// TwinCAT 3 PLC project PLC_Ladder_Hardware_Integration
// ProgramVersion: 3.1.4024.0
// CompilerDefines: VISU_USEWSTRING
// libraries:
//   Tc2_Math, * (Beckhoff Automation GmbH)
//   Tc2_MC2, * (Beckhoff Automation GmbH)
//   Tc2_NC, * (Beckhoff Automation GmbH)
//   Tc2_Standard, * (Beckhoff Automation GmbH)
//   Tc2_System, * (Beckhoff Automation GmbH)
//   Tc2_Utilities, * (Beckhoff Automation GmbH)
//   Tc3_Module, * (Beckhoff Automation GmbH)
// project tree:
//   / GlobalTextList.TcGTLO (not stored), PlcTask.TcTTO, Visualization Manager.TcVMO (not stored), VISU_TASK.TcTTO
//   GVLs/ GVL.TcGVL, GVLLD.TcGVL
//   POUs/ MAIN.TcPOU, ladder_logic_diagram.TcPOU, Meters_Travelled.TcPOU (not stored), SYSTEM.TcPOU, Safety_Zones.TcDUT (not stored), TP_and_TON_For_timeout.TcPOU
//   VISUs/ Charge_Velocity_Distance.TcVIS (not stored), Header.TcVIS (not stored), ImagePool.TcIPO (not stored), log_file.TcVIS (not stored), MainScreen.TcVIS (not stored), Nav.TcVIS (not stored), Nav_1.TcVIS (not stored), Safty_Zones_and_Modes.TcVIS (not stored)
// real-time tasks:
//   TASK PlcTask: cycle T#10ms, priority 20, ADS port 350
//   TASK VISU_TASK: cycle T#200000us, priority 30, ADS port 351
// motion (NC):
//   TASK NC-Task 1 SAF: cycle T#2ms, priority 4, ADS port 501
//   TASK NC-Task 1 SVB: cycle T#10ms, priority 8, ADS port 511
//   AXIS Axis 1 (id 1)
//     Dynamic: Acceleration=2181.51, Deceleration=2181.51, Jerk=6544.55
//     Velo: RefSearch=14.5434333333333, RefSync=14.5434333333333, SlowManual=72.7171666666667, FastManual=436.303, Fast=1454.34333333333, Maximum=1454.34
//     TargetPosControl: Range=20
//     OtherSettings: AllowMotionCmdToSlave=true
//     encoder EncType=19
//       EncPara: ScaleFactorNumerator=15.7, ScaleFactorDenominator=1048576, MaxCount=#xffffffff
//     drive DrvType=16
//       DrvPara: MaxCount=#xffffffff
//         Analog: VeloReferenz=1599.77766666667, VeloScale=32, TorqueSetpointScale=10, ScaleFactorActTorque=0.1
//         TimeComp: TaskDelayCycles=1
//     controller CtrType=1
//       CtrPara: PriorControlFactor=1
//         PosDiffControl: Range=40000
//         Observer: BandWidth=20
//   AXIS Axis 2 (id 2)
//     Dynamic: Acceleration=2181.515, Deceleration=2181.515, Jerk=6544.545
//     Velo: RefSearch=14.5434333333333, RefSync=14.5434333333333, SlowManual=72.7171666666667, FastManual=436.303, Fast=1454.34333333333, Maximum=1454.34333333333
//     TargetPosControl: Range=20
//     OtherSettings: AllowMotionCmdToSlave=true
//     encoder EncType=19
//       EncPara: ScaleFactorNumerator=15.7, ScaleFactorDenominator=1048576, MaxCount=#xffffffff
//     drive DrvType=16
//       DrvPara: MaxCount=#xffffffff
//         Analog: VeloReferenz=1599.77766666667, VeloScale=32, TorqueSetpointScale=10, ScaleFactorActTorque=0.1
//         TimeComp: TaskDelayCycles=1
//     controller CtrType=1
//       CtrPara: PriorControlFactor=1
//         PosDiffControl: Range=40000
//         Observer: BandWidth=20
//   AXIS Axis 3 (id 3)
//     Dynamic: Acceleration=8031.31, Deceleration=8031.31, Jerk=24093.9
//     Velo: RefSearch=53.5420666666667, RefSync=53.5420666666667, SlowManual=267.710333333333, FastManual=1606.262, Fast=5354.20666666667, Maximum=5354.21
//     OtherSettings: AllowMotionCmdToSlave=true
//     encoder EncType=19
//       EncPara: ScaleFactorNumerator=57.8, ScaleFactorDenominator=1048576, MaxCount=#xffffffff
//     drive DrvType=16
//       DrvPara: MaxCount=#xffffffff
//         Analog: VeloReferenz=5889.62733333333, VeloScale=32, TorqueSetpointScale=10, ScaleFactorActTorque=0.1
//         TimeComp: TaskDelayCycles=1
//     controller CtrType=1
//       CtrPara: PriorControlFactor=1
//         PosDiffControl: Range=4000
//         Observer: BandWidth=20
// variable links:
//   PLC_Ladder_Hardware_Integration/PLC_Ladder_Hardware_Integration Instance <-> NC-Task 1 SAF/Axes/Axis 1
//     PlcTask Inputs/MAIN.AxisB.NcToPlc <-> Outputs/ToPlc
//     PlcTask Outputs/MAIN.AxisB.PlcToNc <-> Inputs/FromPlc
//   PLC_Ladder_Hardware_Integration/PLC_Ladder_Hardware_Integration Instance <-> NC-Task 1 SAF/Axes/Axis 2
//     PlcTask Inputs/MAIN.AxisA.NcToPlc <-> Outputs/ToPlc
//     PlcTask Outputs/MAIN.AxisA.PlcToNc <-> Inputs/FromPlc

CONFIGURATION PLC_Ladder_Hardware_Integration
    RESOURCE PLC ON TwinCAT3
        TASK PlcTask(INTERVAL := T#10ms, PRIORITY := 20);
        TASK VISU_TASK(INTERVAL := T#200000us, PRIORITY := 30);
        PROGRAM MAIN WITH PlcTask : MAIN;
        PROGRAM VisuElems_Visu_Prg WITH VISU_TASK : VisuElems.Visu_Prg;
    END_RESOURCE
END_CONFIGURATION

// ---- GVLs/GVL.TcGVL
{attribute 'qualified_only'}
VAR_GLOBAL
	
	GetLocalSystemTime : FB_LocalSystemTime;
	SystemDateTime : STRING;
	SystemDate : STRING;
	SystemTime : STRING;
	SystemSeconds : STRING;
END_VAR

// ---- GVLs/GVLLD.TcGVL
{attribute 'qualified_only'}
VAR_GLOBAL
	
//Input Variables 
ONOFF_Buton               AT %I* : BOOL;
Manual_Stop_Buton         AT %I* : BOOL;
Manual_Mode_Buton         AT %I* : BOOL;
Autonomous_Mode_Buton     AT %I* : BOOL;
Lock_Mode_Buton           AT %I* : BOOL;
Clear_Reset_Buton         AT %I* : BOOL;
Resume_Buton              AT %I* : BOOL;
view_safety               AT %I* : BOOL;


//Output Variables 
Brake                     AT %Q* : BOOL;  
Kontak                    AT %Q* : BOOL;
Front_White_Zone          AT %Q* : BOOL;
Front_Red_Zone            AT %Q* : BOOL;
Front_Purple_Zone         AT %Q* : BOOL;
Front_Grey_Pink_Zone      AT %Q* : BOOL;
Robot_Clear_Lidar         AT %Q* : BOOL;
Robot_Manual_Mode         AT %Q* : BOOL;
Robot_Autonomous_Mode     AT %Q* : BOOL;
Robot_Lock_Mode           AT %Q* : BOOL;
Robot_Mode_Run            AT %Q* : BOOL;
lift_up_Q                 AT %Q* : BOOL;
lift_down_Q            	  AT %Q* : BOOL;
zone_1                    AT %Q* : BOOL;
zone_2                    AT %Q* : BOOL;
zone_3                    AT %Q* : BOOL;
zone_4                    AT %Q* : BOOL;
zone_5                    AT %Q* : BOOL;
zone_6                    AT %Q* : BOOL;
auto_charge_signal        AT %Q* : BOOL;

//Memery Variables 

System_Trig               AT %M* : BOOL;
System_Set                AT %M* : BOOL;
Memory_Set		          AT %M* : BOOL;
White                     AT %M* : BOOL;
Red                       AT %M* : BOOL;
Purple                    AT %M* : BOOL;
Grey_Pink                 AT %M* : BOOL;
Lock_Mode_Reset           AT %M* : BOOL;
lift_up           		  AT %M* : BOOL;
lift_down				  AT %M* : BOOL;
lift_stop				  AT %M* : BOOL;
elavator_up				  AT %M* : BOOL;
elavator_down			  AT %M* : BOOL;
auto_charge_on            AT %M* : BOOL;
auto_charge_off           AT %M* : BOOL;
view_safety_state         AT %M* : BOOL;

first_read		          AT %M* : BOOL;
second_read               AT %M* : BOOL;








	real_trigger: BOOL;
END_VAR

// ---- POUs/MAIN.TcPOU
PROGRAM MAIN
VAR
	Lidar_zones:  Safety_Zones; 
	encoderPosition AT  %I* : UDINT;
	actualAxisPosition AT  %I* : LREAL;
	actualAxisPositionA AT  %I* : LREAL;
	Left_Encoder : LREAL;
	Right_Encoder : LREAL;
	setPositionA AT  %I* : LREAL ;
	setPositionB AT  %I* : LREAL ;
	AxisB : AXIS_REF; //left Motor
	AxisA : AXIS_REF; //Right Motor
	AxisC : AXIS_REF; //Roller Axis
	timer : TON;
	// Motor 1
	McPower : MC_Power;
	McReset : MC_Reset;
	McJogging : MC_Jog;
	McVelocity : MC_MoveVelocity;
	McStop :  MC_Stop;
	McHalt : MC_Halt;
	McSetPositionA: MC_SetPosition;
	McSetPosition: MC_SetPosition;
	McPosition : MC_ReadActualPosition;
	McPositionA : MC_ReadActualPosition;
	McRelativeVelocity : MC_MoveRelative;
	

	// Motor 2
	McPowerA : MC_Power;
	McResetA : MC_Reset;
	McJoggingA : MC_Jog;
	McVelocityA : MC_MoveVelocity;
	McStopA :  MC_Stop;
	McHaltA : MC_Halt;
	
	CppVelocityValue : DINT;
	CppVelocityCmd : DINT;
	RightVelocityValue : REAL;
	LeftVelocityValue : REAL;
	RightVelocityCmd : REAL;
	LeftVelocityCmd : REAL;
	RollerVelocityValue : REAL;
	RollerVelocityCmd : REAL;
	RightVelocity_meters : REAL;
	LeftVelocity_meters : REAL;
	acc : REAL:=0;
	dcc : REAL:=0;
	jk	: REAL:=0;
	myvelocity : DINT;
	cppvar AT %I* : BOOL;
	pypositive AT %I* : BOOL;
	pynegative AT %I* : BOOL;
	pyturnright AT %I* : BOOL;
	pyturnleft AT %I* : BOOL;
	state : DINT;
	stop AT %I* : BOOL;
	fright AT %I* : BOOL;
	bright AT %I* : BOOL;
	fleft AT %I* : BOOL;
	bleft AT %I* : BOOL;
	roller_forward     AT %I* : BOOL;
	roller_backwrad    AT %I* : BOOL;
	ChargeSignal       AT %Q* : BOOL;
	Lift_UP            AT %Q* : BOOL:= FALSE;
	Lift_DOWN          AT %Q* : BOOL;
	Lift_UP_Signal	   AT %M* : BOOL;
	Lift_DOWN_Signal   AT %M* : BOOL;
	Lift_Stop          AT %M* : BOOL;
	FrontLidarWarning  AT %I* : BOOL;
	BackLidarWarning   AT %I* : BOOL;

	stopvalue : BOOL;
	Acceleration: LREAL;
	Options: INT;
	nVAR: REAL;
	
	time_first_read : INT;
	time_second_read : INT;
	//Lidar Zones
	zon_1_set          AT %M* : BOOL; 
	zon_2_set          AT %M* : BOOL; 
	zon_3_set          AT %M* : BOOL; 
	zon_4_set          AT %M* : BOOL; 
	zon_5_set          AT %M* : BOOL; 
	zon_6_set          AT %M* : BOOL;    
	
	
	
END_VAR

SYSTEM();
Meters_Travelled();
Ladder_Logic_Diagram();
encoderPosition;
TP_and_TON_For_timeout();

IF GVLLD.first_read THEN	
time_first_read := STRING_TO_INT (GVL.SystemSeconds);
END_IF
IF GVLLD.second_read THEN	
time_second_read := STRING_TO_INT (GVL.SystemSeconds);
END_IF

// Axis B Left Motor
AxisB.ReadStatus();
McPower(Axis:=AxisB,Enable := TRUE,Enable_Positive := TRUE, Enable_Negative := TRUE);
McSetPosition(Axis:= AxisB,Execute:= TRUE, Position := setPositionA);
McPosition(Axis := AxisB,Enable := TRUE );
actualAxisPosition := McPosition.Position;
Left_Encoder := actualAxisPosition ;

// Axis A Right Motor
AxisA.ReadStatus();
McPowerA(Axis:=AxisA,Enable := TRUE,Enable_Positive := TRUE, Enable_Negative := TRUE);
McSetPositionA(Axis:= AxisA,Execute:= TRUE, Position := setPositionB);
McPositionA(Axis := AxisA,Enable := TRUE );
actualAxisPositionA := McPositionA.Position;
Right_Encoder := actualAxisPositionA ;


CppVelocityCmd := CppVelocityValue;
RightVelocity_meters := RightVelocityCmd /1000 ;
LeftVelocity_meters := LeftVelocityCmd / 1000 ;
IF NOT GVLLD.view_safety THEN
	RightVelocityCmd := 0;
	LeftVelocityCmd := 0;
	RollerVelocityCmd := 0;
	ELSE IF NOT FrontLidarWarning OR NOT BackLidarWarning THEN
		RightVelocityCmd := RightVelocityValue * 0.9;
		LeftVelocityCmd := LeftVelocityValue * 0.9;
	ELSE IF FrontLidarWarning OR BackLidarWarning THEN
		RightVelocityCmd := RightVelocityValue;
		LeftVelocityCmd := LeftVelocityValue;
		RollerVelocityCmd := RollerVelocityValue;
		END_IF
	END_IF
END_IF

stopvalue := stop;



CASE state OF 
	0: 	
		state := 10;
	10: 
	
		McReset(Axis := AxisB,Execute := TRUE);
		McResetA(Axis := AxisA,Execute := TRUE);
		IF McReset.Done AND McResetA.Done  THEN
			state := 20;
		ELSIF NOT McReset.Done OR NOT McResetA.Done THEN 
			McReset(Axis := AxisB,Execute := FALSE);
			McResetA(Axis := AxisA,Execute := FALSE);
			McReset(Axis := AxisB,Execute := TRUE);
			McResetA(Axis := AxisA,Execute := TRUE);
			state := 20;
		END_IF
		
	20: 
	
		McPowerA(Axis:=AxisA,Enable := TRUE,Enable_Positive := TRUE, Enable_Negative := TRUE);
		McPower(Axis:=AxisB,Enable := TRUE,Enable_Positive := TRUE, Enable_Negative := TRUE);
		IF McPower.Status AND McPowerA.Status THEN
			McReset(Axis := AxisB,Execute := TRUE);
			McResetA(Axis := AxisA,Execute := TRUE);
			IF McReset.Done AND McResetA.Done  THEN
				state :=50;
			ELSIF NOT McReset.Done OR NOT McResetA.Done THEN 
				McReset(Axis := AxisB,Execute := FALSE);
				McResetA(Axis := AxisA,Execute := FALSE);
				McReset(Axis := AxisB,Execute := TRUE);
				McResetA(Axis := AxisA,Execute := TRUE);
				state :=50;
			END_IF
		END_IF
		
	
	//CPP Function Block
//	40: 
		
//		McVelocityA (Axis:= AxisA,
//					Execute := cppvar,
//					Velocity := CppVelocityCmd,
//						Acceleration := acc,
//						Deceleration := dcc,
//						Jerk := jk,
//					Direction := MC_Direction.MC_Positive_Direction ) ;
//		McVelocity (Axis:= AxisB,
//					Execute := cppvar,
//					Velocity := CppVelocityCmd,
//						Acceleration := acc,
//						Deceleration := dcc,
//						Jerk := jk,
//					Direction := MC_Direction.MC_Positive_Direction ) ;
//		McVelocityA (Axis:= AxisA,
//					Execute := cppvar,
//					Velocity := CppVelocityCmd,
//						Acceleration := acc,
//						Deceleration := dcc,
//						Jerk := jk,
//					Direction := MC_Direction.MC_Negative_Direction ) ;
//		McVelocity (Axis:= AxisB,
//					Execute := cppvar,
//					Velocity := CppVelocityCmd,
//						Acceleration := acc,
//						Deceleration := dcc,
//						Jerk := jk,
//					Direction := MC_Direction.MC_Negative_Direction ) ;
//		IF stopvalue THEN
//			McVelocity(Axis := AxisB, Execute := FALSE); 
//			McVelocityA(Axis := AxisA, Execute := FALSE); 
//			state := 900;
//		END_IF
//		IF fright OR fleft OR bright OR bleft THEN 
//			McVelocity(Axis := AxisB, Execute := FALSE);
//			McVelocityA(Axis := AxisA, Execute := FALSE);
//			state := 50;
//		END_IF
		
		
	//Python Function Block
	50: 
		// POSİTİVE
		IF AxisA.Status.Error OR AxisB.Status.Error THEN 
			McReset(Axis := AxisB,Execute := FALSE);
			McResetA(Axis := AxisA,Execute := FALSE);
			McReset(Axis := AxisB,Execute := TRUE);
			McResetA(Axis := AxisA,Execute := TRUE);
//			state :=0;
		END_IF
		IF stopvalue THEN
			
			McVelocity(Axis := AxisB, Execute := FALSE); 
			McVelocityA(Axis := AxisA, Execute := FALSE);
			state := 900;
		END_IF
		IF GVLLD.auto_charge_signal THEN   
   			McVelocity(Axis := AxisB, Execute := FALSE);    
			McVelocityA(Axis := AxisA, Execute := FALSE);
  			state := 400;  
		END_IF
		
		McVelocityA (Axis:= AxisA,
						Execute := fright,
						Velocity := RightVelocityCmd,
						Acceleration := acc,
						Deceleration := dcc,
						Jerk := jk,
						Direction := MC_Direction.MC_Positive_Direction ) ;
		McVelocityA (Axis:= AxisA,
						Execute := bright,
						Velocity := RightVelocityCmd,
						Acceleration := acc,
						Deceleration := dcc,
						Jerk := jk,
						Direction := MC_Direction.MC_Negative_Direction ) ;
		McVelocity (Axis:= AxisB,
						Execute := fleft,
						Velocity := LeftVelocityCmd,
						Acceleration := acc,
						Deceleration := dcc,
						Jerk := jk,
						Direction := MC_Direction.MC_Positive_Direction ) ;
		McVelocity (Axis:= AxisB,
						Execute := bleft,
						Velocity := LeftVelocityCmd,
						Acceleration := acc,
						Deceleration := dcc,
						Jerk := jk,
						Direction := MC_Direction.MC_Negative_Direction ) ;
// Roller Velocity Blocks
//Forward
//		MC_MoveContinuousRelative(Axis:=AxisC,
//								Execute:= roller_forward,
//								Distance:= 5000,
//								Velocity:= 1000,
//								EndVelocity:= 0,
//								Acceleration:= acc,
//								Deceleration:= dcc,
//								Jerk:= jk);
////Backward 
//		MC_MoveContinuousRelative(Axis:=AxisC,
//								Execute:= roller_backwrad,
//								Distance:= 5000,
//								Velocity:= RollerVelocityValue,
//								EndVelocity:= 0,
//								Acceleration:= acc,
//								Deceleration:= dcc,
//								Jerk:= jk);
		IF cppvar THEN 
			McVelocity(Axis := AxisB, Execute := FALSE);
			McVelocityA(Axis := AxisA, Execute := FALSE);
			state := 40;
		END_IF
	400:  
		IF AxisA.Status.Error OR AxisB.Status.Error THEN 
		   	McReset(Axis := AxisB,Execute := FALSE);   
			McResetA(Axis := AxisA,Execute := FALSE);
		   	McReset(Axis := AxisB,Execute := TRUE);   
			McResetA(Axis := AxisA,Execute := TRUE);
  		END_IF
    	McStop(Axis := AxisB, Execute := TRUE);
  		McStopA(Axis := AxisA, Execute := TRUE);  
  		IF NOT GVLLD.auto_charge_signal THEN   
			McStop(Axis := AxisB, Execute := FALSE); 
			McVelocity(Axis := AxisB, Execute := FALSE);    
			McStopA(Axis := AxisA, Execute := FALSE); 
			McVelocityA(Axis := AxisA, Execute := FALSE);    
			state := 50;
  		END_IF
	900:
		IF AxisA.Status.Error OR AxisB.Status.Error THEN 
			McReset(Axis := AxisB,Execute := FALSE);
			McResetA(Axis := AxisA,Execute := FALSE);
			McReset(Axis := AxisB,Execute := TRUE);
			McResetA(Axis := AxisA,Execute := TRUE);
		END_IF
		McStop(Axis := AxisB, Execute := TRUE);
		McStopA(Axis := AxisA, Execute := TRUE);
		IF fright OR fleft OR bright OR bleft OR pyturnleft OR cppvar THEN
			McStop(Axis := AxisB, Execute := FALSE); 
			McVelocity(Axis := AxisB, Execute := FALSE); 
			McStopA(Axis := AxisA, Execute := FALSE); 
			McVelocityA(Axis := AxisA, Execute := FALSE); 
			state := 50;
		END_IF
		
		
		
END_CASE

END_PROGRAM

// ---- POUs/SYSTEM.TcPOU
PROGRAM SYSTEM
VAR
END_VAR

GVL.GetLocalSystemTime(
	sNetID := ,
	bEnable := TRUE,
	dwCycle := 1,
	dwOpt:= ,
	tTimeout:= ,
	bValid =>,
	systemTime=>,
	tzID=>);
	
GVL.SystemDateTime := SYSTEMTIME_TO_STRING(GVL.GetLocalSystemTime.systemTime);
GVL.SystemDate := MID(STR:= GVL.SystemDateTime,LEN:=10,POS:=1);
GVL.SystemTime := MID(STR:= GVL.SystemDateTime,LEN:=8,POS:=12);
GVL.SystemSeconds := MID(STR:= GVL.SystemDateTime,LEN:=2,POS:=18);

END_PROGRAM

// ---- POUs/ladder_logic_diagram.TcPOU
PROGRAM ladder_logic_diagram 
VAR
	t2s: TIME := TIME#3S;
	t0s: TIME := TIME#0S;
	Timer: TON;
	input : BOOL;
	output : BOOL; 
	TON_Reset: TON;
	TON_set: TON;
	TON_0: TON;
	TON_Trig: TON;
	TON_Autonomous: TON;
	TON_Manual: TON;
	TON_Lock: TON;
	Robot_Mode_Timer: TON;
	liftUP: TON;
	liftDOWN: TON;

	T: TIME;
	Activate_time_read: BOOL;
	TON_1: TON;
	first_read_triggerd: BOOL;
	TON_2: TON;
	second_read_triggerd: BOOL;
	TON_3: TON;
	TON_4: TON;
	TON_5: TON;
	trig_1: BOOL;
	TP_0: TP;
	TP_1: TP;
	trig_2: BOOL;
	load_button: BOOL;
	TON_6: TON;
	load_active: BOOL;
	TON_7: TON;
END_VAR
VAR // added by the converter: edge detectors and wires of the graphical bodies
    _rt1 : R_TRIG;
    _w1 : BOOL;
END_VAR

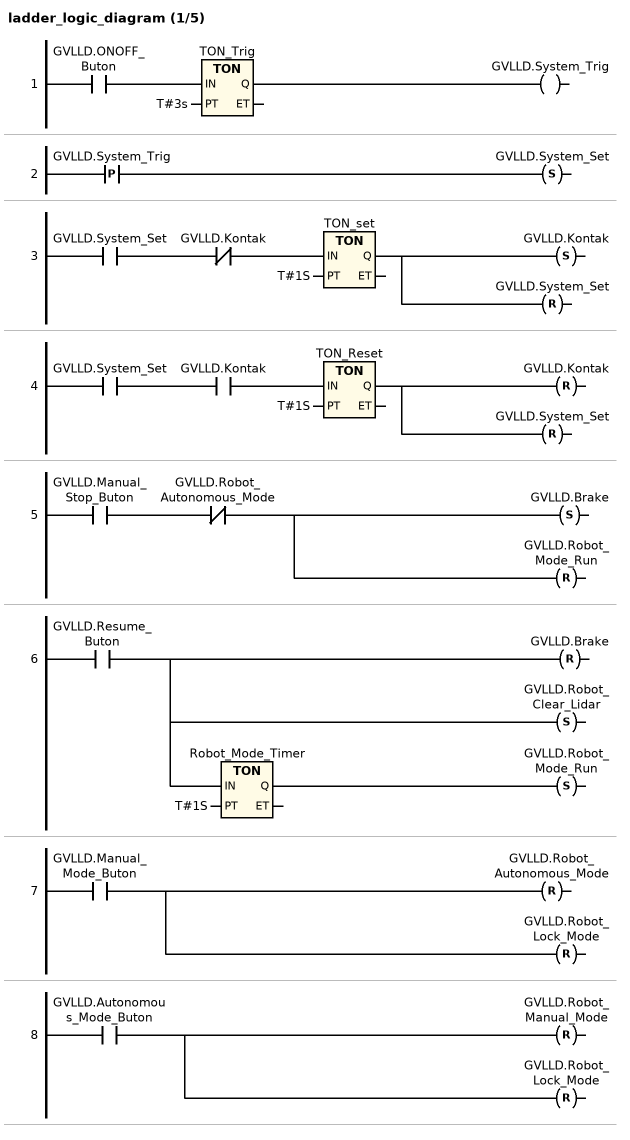
// NETWORK 1
TON_Trig(IN := GVLLD.ONOFF_Buton, PT := T#3s); // TON
GVLLD.System_Trig := TON_Trig.Q;

// NETWORK 2
_rt1(CLK := GVLLD.System_Trig);
GVLLD.System_Set S= _rt1.Q;

// NETWORK 3
TON_set(IN := GVLLD.System_Set AND NOT GVLLD.Kontak, PT := T#1S); // TON
GVLLD.Kontak S= TON_set.Q;
GVLLD.System_Set R= TON_set.Q;

// NETWORK 4
TON_Reset(IN := GVLLD.System_Set AND GVLLD.Kontak, PT := T#1S); // TON
GVLLD.Kontak R= TON_Reset.Q;
GVLLD.System_Set R= TON_Reset.Q;

// NETWORK 5
_w1 := GVLLD.Manual_Stop_Buton AND NOT GVLLD.Robot_Autonomous_Mode;
GVLLD.Brake S= _w1;
GVLLD.Robot_Mode_Run R= _w1;

// NETWORK 6
GVLLD.Brake R= GVLLD.Resume_Buton;
GVLLD.Robot_Clear_Lidar S= GVLLD.Resume_Buton;
Robot_Mode_Timer(IN := GVLLD.Resume_Buton, PT := T#1S); // TON
GVLLD.Robot_Mode_Run S= Robot_Mode_Timer.Q;

// NETWORK 7
GVLLD.Robot_Autonomous_Mode R= GVLLD.Manual_Mode_Buton;
GVLLD.Robot_Lock_Mode R= GVLLD.Manual_Mode_Buton;

// NETWORK 8
GVLLD.Robot_Manual_Mode R= GVLLD.Autonomous_Mode_Buton;
GVLLD.Robot_Lock_Mode R= GVLLD.Autonomous_Mode_Buton;

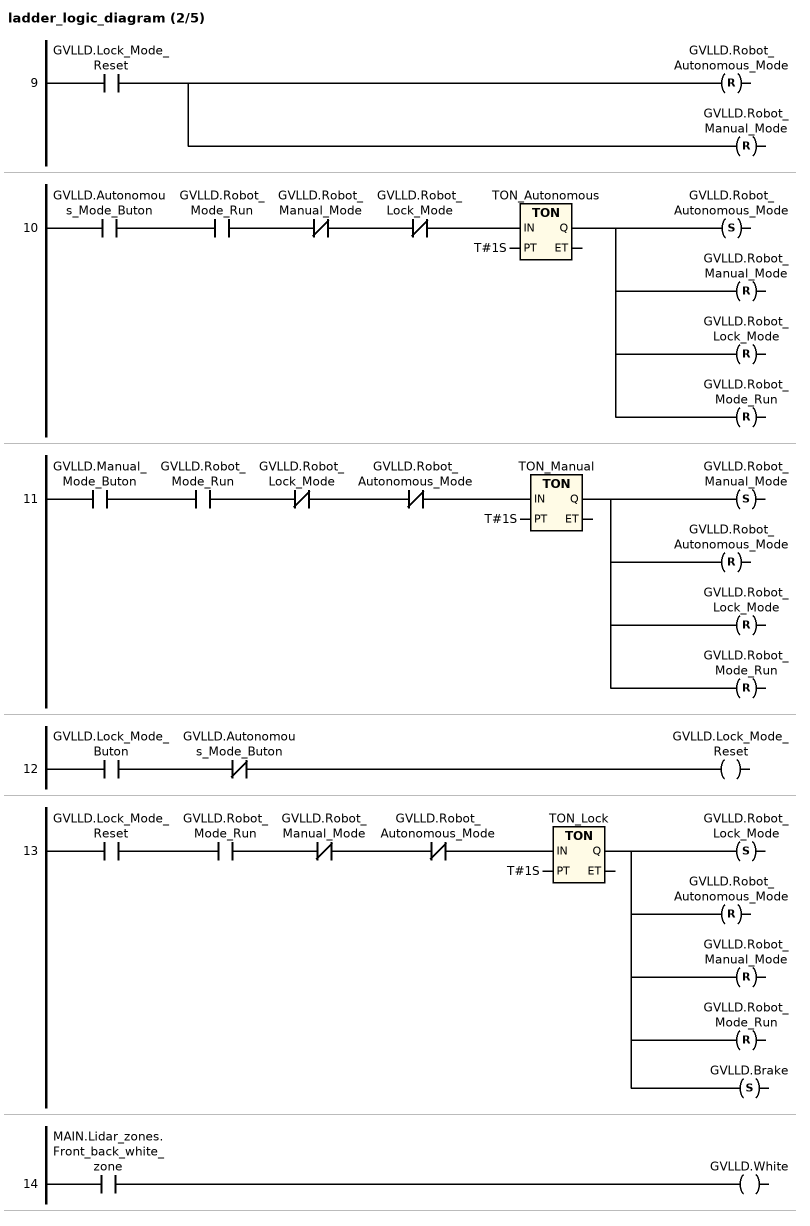
// NETWORK 9
GVLLD.Robot_Autonomous_Mode R= GVLLD.Lock_Mode_Reset;
GVLLD.Robot_Manual_Mode R= GVLLD.Lock_Mode_Reset;

// NETWORK 10
TON_Autonomous(IN := GVLLD.Autonomous_Mode_Buton AND GVLLD.Robot_Mode_Run AND NOT GVLLD.Robot_Manual_Mode AND NOT GVLLD.Robot_Lock_Mode, PT := T#1S); // TON
GVLLD.Robot_Autonomous_Mode S= TON_Autonomous.Q;
GVLLD.Robot_Manual_Mode R= TON_Autonomous.Q;
GVLLD.Robot_Lock_Mode R= TON_Autonomous.Q;
GVLLD.Robot_Mode_Run R= TON_Autonomous.Q;

// NETWORK 11
TON_Manual(IN := GVLLD.Manual_Mode_Buton AND GVLLD.Robot_Mode_Run AND NOT GVLLD.Robot_Lock_Mode AND NOT GVLLD.Robot_Autonomous_Mode, PT := T#1S); // TON
GVLLD.Robot_Manual_Mode S= TON_Manual.Q;
GVLLD.Robot_Autonomous_Mode R= TON_Manual.Q;
GVLLD.Robot_Lock_Mode R= TON_Manual.Q;
GVLLD.Robot_Mode_Run R= TON_Manual.Q;

// NETWORK 12
GVLLD.Lock_Mode_Reset := GVLLD.Lock_Mode_Buton AND NOT GVLLD.Autonomous_Mode_Buton;

// NETWORK 13
TON_Lock(IN := GVLLD.Lock_Mode_Reset AND GVLLD.Robot_Mode_Run AND NOT GVLLD.Robot_Manual_Mode AND NOT GVLLD.Robot_Autonomous_Mode, PT := T#1S); // TON
GVLLD.Robot_Lock_Mode S= TON_Lock.Q;
GVLLD.Robot_Autonomous_Mode R= TON_Lock.Q;
GVLLD.Robot_Manual_Mode R= TON_Lock.Q;
GVLLD.Robot_Mode_Run R= TON_Lock.Q;
GVLLD.Brake S= TON_Lock.Q;

// NETWORK 14
GVLLD.White := MAIN.Lidar_zones.Front_back_white_zone;

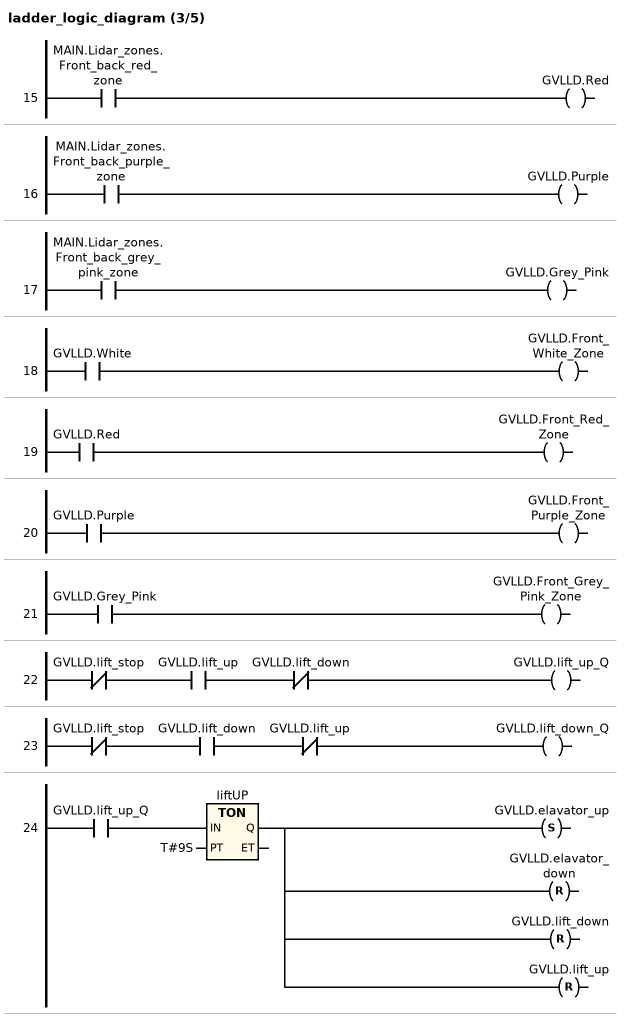
// NETWORK 15
GVLLD.Red := MAIN.Lidar_zones.Front_back_red_zone;

// NETWORK 16
GVLLD.Purple := MAIN.Lidar_zones.Front_back_purple_zone;

// NETWORK 17
GVLLD.Grey_Pink := MAIN.Lidar_zones.Front_back_grey_pink_zone;

// NETWORK 18
GVLLD.Front_White_Zone := GVLLD.White;

// NETWORK 19
GVLLD.Front_Red_Zone := GVLLD.Red;

// NETWORK 20
GVLLD.Front_Purple_Zone := GVLLD.Purple;

// NETWORK 21
GVLLD.Front_Grey_Pink_Zone := GVLLD.Grey_Pink;

// NETWORK 22
GVLLD.lift_up_Q := NOT GVLLD.lift_stop AND GVLLD.lift_up AND NOT GVLLD.lift_down;

// NETWORK 23
GVLLD.lift_down_Q := NOT GVLLD.lift_stop AND GVLLD.lift_down AND NOT GVLLD.lift_up;

// NETWORK 24
liftUP(IN := GVLLD.lift_up_Q, PT := T#9S); // TON
GVLLD.elavator_up S= liftUP.Q;
GVLLD.elavator_down R= liftUP.Q;
GVLLD.lift_down R= liftUP.Q;
GVLLD.lift_up R= liftUP.Q;

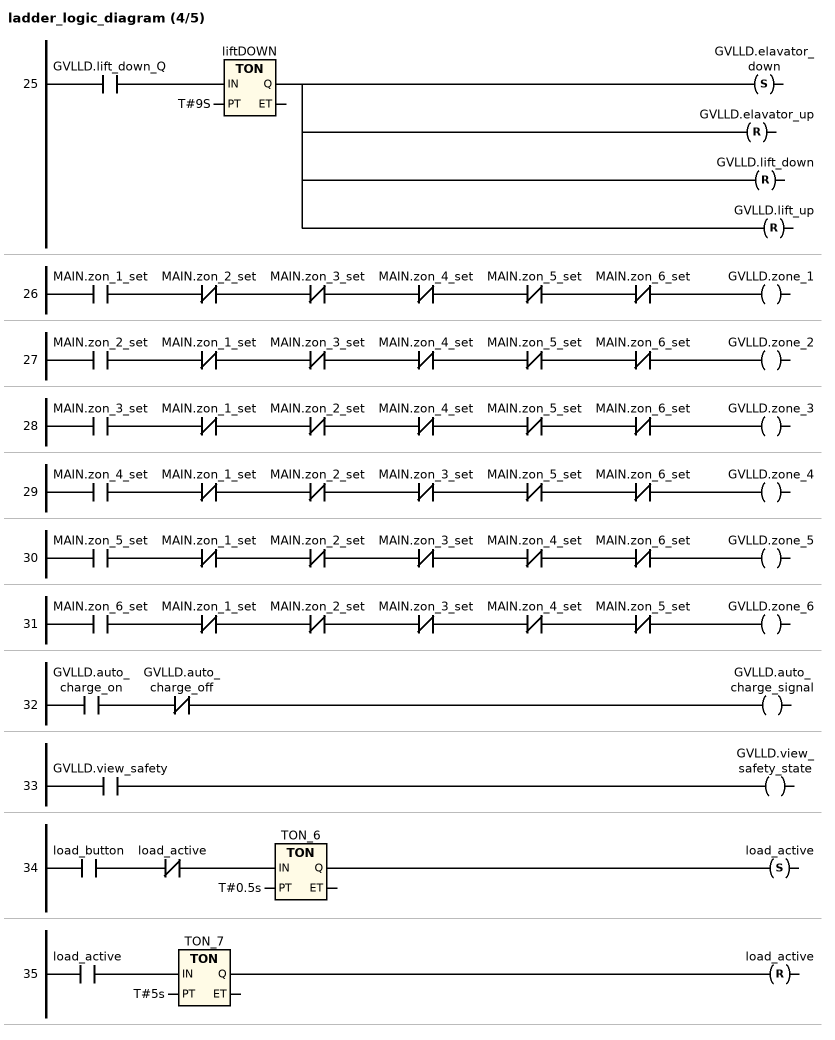
// NETWORK 25
liftDOWN(IN := GVLLD.lift_down_Q, PT := T#9S); // TON
GVLLD.elavator_down S= liftDOWN.Q;
GVLLD.elavator_up R= liftDOWN.Q;
GVLLD.lift_down R= liftDOWN.Q;
GVLLD.lift_up R= liftDOWN.Q;

// NETWORK 26
GVLLD.zone_1 := MAIN.zon_1_set AND NOT MAIN.zon_2_set AND NOT MAIN.zon_3_set AND NOT MAIN.zon_4_set AND NOT MAIN.zon_5_set AND NOT MAIN.zon_6_set;

// NETWORK 27
GVLLD.zone_2 := MAIN.zon_2_set AND NOT MAIN.zon_1_set AND NOT MAIN.zon_3_set AND NOT MAIN.zon_4_set AND NOT MAIN.zon_5_set AND NOT MAIN.zon_6_set;

// NETWORK 28
GVLLD.zone_3 := MAIN.zon_3_set AND NOT MAIN.zon_1_set AND NOT MAIN.zon_2_set AND NOT MAIN.zon_4_set AND NOT MAIN.zon_5_set AND NOT MAIN.zon_6_set;

// NETWORK 29
GVLLD.zone_4 := MAIN.zon_4_set AND NOT MAIN.zon_1_set AND NOT MAIN.zon_2_set AND NOT MAIN.zon_3_set AND NOT MAIN.zon_5_set AND NOT MAIN.zon_6_set;

// NETWORK 30
GVLLD.zone_5 := MAIN.zon_5_set AND NOT MAIN.zon_1_set AND NOT MAIN.zon_2_set AND NOT MAIN.zon_3_set AND NOT MAIN.zon_4_set AND NOT MAIN.zon_6_set;

// NETWORK 31
GVLLD.zone_6 := MAIN.zon_6_set AND NOT MAIN.zon_1_set AND NOT MAIN.zon_2_set AND NOT MAIN.zon_3_set AND NOT MAIN.zon_4_set AND NOT MAIN.zon_5_set;

// NETWORK 32
GVLLD.auto_charge_signal := GVLLD.auto_charge_on AND NOT GVLLD.auto_charge_off;

// NETWORK 33
GVLLD.view_safety_state := GVLLD.view_safety;

// NETWORK 34
TON_6(IN := load_button AND NOT load_active, PT := T#0.5s); // TON
load_active S= TON_6.Q;

// NETWORK 35
TON_7(IN := load_active, PT := T#5s); // TON
load_active R= TON_7.Q;

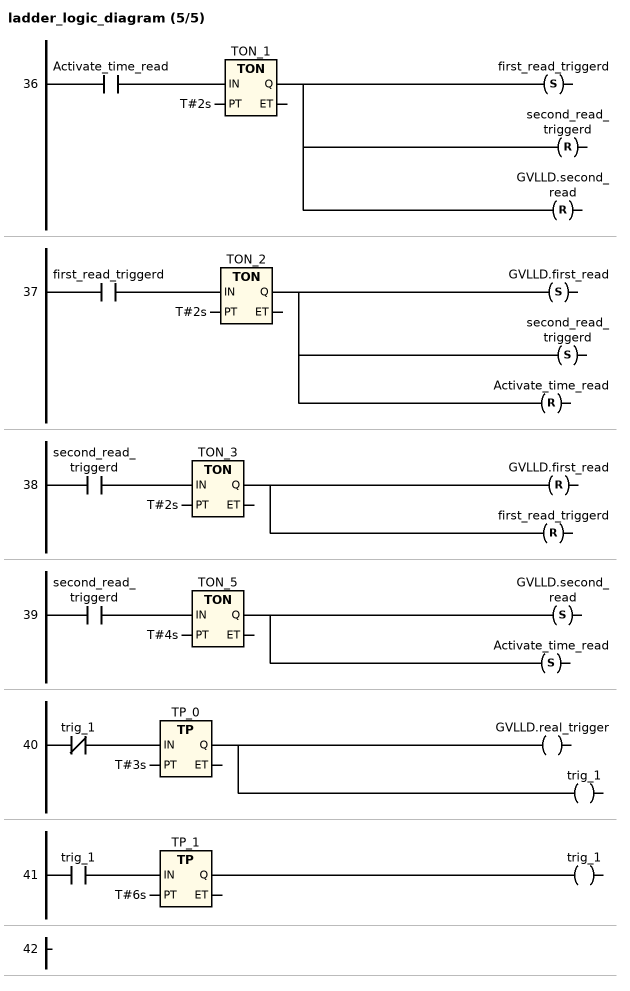
// NETWORK 36
TON_1(IN := Activate_time_read, PT := T#2s); // TON
first_read_triggerd S= TON_1.Q;
second_read_triggerd R= TON_1.Q;
GVLLD.second_read R= TON_1.Q;

// NETWORK 37
TON_2(IN := first_read_triggerd, PT := T#2s); // TON
GVLLD.first_read S= TON_2.Q;
second_read_triggerd S= TON_2.Q;
Activate_time_read R= TON_2.Q;

// NETWORK 38
TON_3(IN := second_read_triggerd, PT := T#2s); // TON
GVLLD.first_read R= TON_3.Q;
first_read_triggerd R= TON_3.Q;

// NETWORK 39
TON_5(IN := second_read_triggerd, PT := T#4s); // TON
GVLLD.second_read S= TON_5.Q;
Activate_time_read S= TON_5.Q;

// NETWORK 40
TP_0(IN := NOT trig_1, PT := T#3s); // TP
GVLLD.real_trigger := TP_0.Q;
trig_1 := TP_0.Q;

// NETWORK 41
TP_1(IN := trig_1, PT := T#6s); // TP
trig_1 := TP_1.Q;

// NETWORK 42

END_PROGRAM

// ---- POUs/TP_and_TON_For_timeout.TcPOU
PROGRAM TP_and_TON_For_timeout
VAR
	TP_1_trigger: BOOL;
	TP_1: TP;
	Trig_TON_1: BOOL;
	TON_1: TON;
	TP_2_trigger: BOOL;
	TP_2: TP;
	Trig_TON_2: BOOL;
	TON_2: TON;
END_VAR

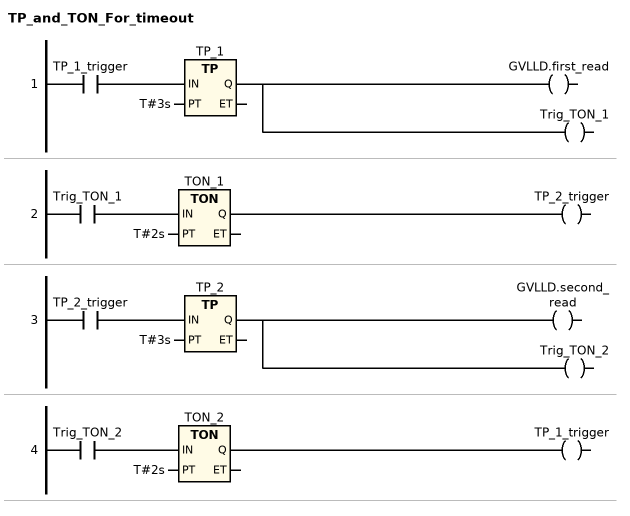
// NETWORK 1
TP_1(IN := TP_1_trigger, PT := T#3s); // TP
GVLLD.first_read := TP_1.Q;
Trig_TON_1 := TP_1.Q;

// NETWORK 2
TON_1(IN := Trig_TON_1, PT := T#2s); // TON
TP_2_trigger := TON_1.Q;

// NETWORK 3
TP_2(IN := TP_2_trigger, PT := T#3s); // TP
GVLLD.second_read := TP_2.Q;
Trig_TON_2 := TP_2.Q;

// NETWORK 4
TON_2(IN := Trig_TON_2, PT := T#2s); // TON
TP_1_trigger := TON_2.Q;

END_PROGRAM
